TYPE T_ASTRO_CCS_DATA :
STRUCT
	environment :	T_ASTRO_ENVIRONMENT;
	site :			T_ASTRO_SITE_CONSTANTS;
	motion :		T_ASTRO_POLAR_MOTION;
	dut :			LREAL;
	equinox :		LREAL;
	wavelength :	LREAL;
END_STRUCT
END_TYPE

(* stored: Version 1.1.0.1, ProductVersion 3.1.4024.10
   DUT T_ASTRO_CCS_DATA: Id {22a6f6f9-06cd-4b97-800c-e19e17ff92e4} *)
